{attribute 'qualified_only'}
{attribute 'strict'}
TYPE E_MergeType :
(
	NoSlowdown := 0,
	StartFromMergeWaitStatic := 1,
	Decelerating := 2 
);
END_TYPE

(* stored: Version 1.1.0.1, ProductVersion 3.1.4026.8
   DUT E_MergeType: Id {5f2b2829-d5cc-006a-38b4-db1394be2037} *)
